(* CODESYS project FU_sPaddBackLen.xml

Project tree, tasks and I/O mapping:
  function FU_sPaddBackLen [ST]
*)

// FU_sPaddBackLen
//This function padds the back of a string with the given character, the given amount
//If the padd amount plus the string is longer than the output string, the input string will be cut off to make space for the padding
// +-----------+----------+----------+-----------------------------------------------------------------------------------------------------------------------+
// |**Version**|**Author**| **Date** |**Changes**                                                                                                            |
// +-----------+----------+----------+-----------------------------------------------------------------------------------------------------------------------+
// | 1         | NSN      | 04-02-19 | Creation                                                                                                              |
// +-----------+----------+----------+-----------------------------------------------------------------------------------------------------------------------+
FUNCTION FU_sPaddBackLen  : STRING(255)
VAR_INPUT
	sStr		:STRING(255);		//Input String
	wLen		:WORD;				//How much to padd it
	eChar		:EASCII;		//Which character to padd with
END_VAR

FU_sPaddBackLenBIBO(sOut:=FU_sPaddBackLen,sStr:=sStr,wLen:=wLen,wOutSize:=255,eChar:=eChar);

END_FUNCTION
